//{attribute 'qualified_only'}
VAR_GLOBAL
	iVentilatie		AT %Q*	: INT;
	
	bVentUp					: BOOL;
	bVentDown				: BOOL;
END_VAR

(* stored: Version 1.1.0.1
   GVL GVL_Ventilatie: Id {a367bac8-a5e7-4789-ac08-164e37206a9c} *)
